PROGRAM MAIN
VAR
END_VAR

Prog_Arrays();

END_PROGRAM

(* stored: Version 1.1.0.1, ProductVersion 3.1.4024.9
   POU MAIN: Id {ad62ed39-3df3-4e9c-bd06-abfc34e53603}, SpecialFunc None *)
